// SIMATIC S7-200 project (STEP 7-Micro/WIN), CPU 222 CN REL 02.01

SYMBOL_TABLE 
USS_LOW_V        VD1000
USS_HIGH_V       VD1004
USS_TIME_OUT     VW1008
USS_I_LINE       VW1010
USS_DAT_PTR0     VD1012
USS_ACT_DRV0     VD1016
USS_CUR_DRV0     VD1020
USS_P0           V1024.0
USS_REQ_SNT0     V1024.1
USS_RETRY_P0     VB1025
USS_ERR_CODE     VB1026
USS_CS_D0        VD1027
USS_CS_W0        VW1027
USS_CS_W2        VW1029
USS_CS_B0        VB1027
USS_CS_B1        VB1028
USS_POLL_BUF     VB1031
USS_XMT_0        VB1046
USS_XMT_ADR0     VB1049
USS_X_STWD       VD1056
USS_X_BCC        VB1060
USS_X_DW1        VD1047
USS_X_DW5        VD1051
USS_X_DW9        VD1055
USS_X_DB13       VB1059
USS_RCV_BUF0     VB1061
USS_R_STX        VB1062
USS_R_LGE        VB1063
USS_R_ADR        VB1064
USS_R_STWD       VD1071
USS_R_DW1        VD1062
USS_R_DW5        VD1066
USS_R_DW9        VD1070
USS_R_W13        VW1074
USS_STAT_TAB     VB1076
USS_ADR_P0       VB1396
END_SYMBOL_TABLE

// OB1: protected block, not included

// SBR0: protected block, not included

// INT0: protected block, not included

// INT1: protected block, not included
